{attribute 'qualified_only'}
{attribute 'strict'}
TYPE DUT :
(
	off,
	Reset,
	Power,
	Ready,
	Moving
);
END_TYPE

(* stored: Version 1.1.0.1, ProductVersion 3.1.4024.15
   DUT DUT: Id {f2cf7833-5ead-4ee1-93cd-a7d3d2ae6617} *)
